FUNCTION_BLOCK FB_SchmittTriggerConsumer
VAR
    trigger : T1SchmittTrigger_Plc.FB_SchmittTrigger;
    bLastState : BOOL;
END_VAR

trigger(fInput := 0.5);
bLastState := trigger.Step();

END_FUNCTION_BLOCK

(* stored: Version 1.1.0.1
   POU FB_SchmittTriggerConsumer: Id {0575cae4-8b45-4f3b-a43a-366d9af87697}, SpecialFunc None *)
